PROGRAM Alarm_Flag
VAR
END_VAR

// NETWORK 1

END_PROGRAM

(* stored: Version 1.1.0.1, ProductVersion 3.1.4024.0
   POU Alarm_Flag: Id {e25eff55-c5ba-4395-b8fa-f60a021d8a05}, SpecialFunc None *)
